SUBAPPLICATION AS_TO_Q_NumericValue (* AS-Adapter-Wert (z.B. Schrittkettennummer) via AUDI auf ein VT-Zahlenfeld (Q_NumericValue_AUDI) anzeigen. Generisch, Object ID parametrierbar. Schwester-Baustein zu MyLib::sys::SINT_TO_Q_NumericValue (dort direkte SINT-Verdrahtung statt AS-Adapter). *)
  (* Standard: 61499-2 *)
  (* Version 1.0, 2026-09-09, Franz Höpfinger, Meisterschulen am Ostbahnhof, Ausgelagert aus Uebung_039_sub_NumbAnzeig_AS zur Wiederverwendung; u16ObjId zuvor fest importiert (OutputNumber_N1), jetzt als VarDeclaration parametrierbar. *)
  PACKAGE MyLib::sys;
  IMPORT isobus::UT::Q::const::IDs::ID_NULL;
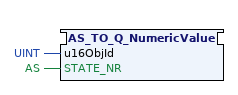
  VAR_INPUT
    u16ObjId : UINT := ID_NULL; (* Object ID *)
  END_VAR
  SOCKETS
    STATE_NR : adapter::types::unidirectional::AS;
  END_SOCKETS
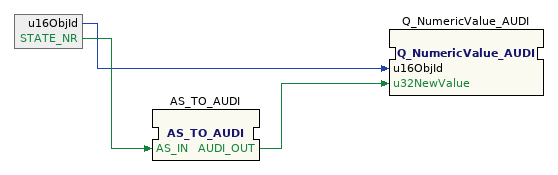
  FBS
    Q_NumericValue_AUDI : isobus::UT::Q::Q_NumericValue_AUDI;
    AS_TO_AUDI : adapter::conversion::unidirectional::AS_TO_AUDI;
  END_FBS
  DATA_CONNECTIONS
    u16ObjId TO Q_NumericValue_AUDI.u16ObjId;
  END_CONNECTIONS
  ADAPTER_CONNECTIONS
    AS_TO_AUDI.AUDI_OUT TO Q_NumericValue_AUDI.u32NewValue;
    STATE_NR TO AS_TO_AUDI.AS_IN;
  END_CONNECTIONS
END_SUBAPPLICATION
